(* IEC 61131-3 sources: Std_PalletMover/Class/_LMCAxisVOVMonitoring, 1 file *)

(* ---- _LMCAxisVOVMonitoring.st ---- *)
// Monitoring time (ms). If a button is not being pressed or released for a this amount of time the connection has been broken
#ifndef LMCAXIS_VOVMonitor_NoReactionTimeLimit
  #define  LMCAXIS_VOVMonitor_NoReactionTimeLimit 1000 ms
#endif

(*!
<Class
	Name               = "_LMCAxisVOVMonitoring"
	Revision           = "1.0"
	RealtimeTask       = "false"
	CyclicTask         = "false"
	BackgroundTask     = "true"
	DefBackground      = "10 ms"
	Sigmatek           = "true"
	OSInterface        = "false"
	HighPriority       = "false"
	Automatic          = "false"
	UpdateMode         = "Prescan"
	IconPath           = ".\Class\_LMCAxisVis\LMCAxis.ico"
	SharedCommandTable = "true"
	Objectsize         = "(284,120)"
	Comment            = "Class used to observe if a move hand button is still actively pressed in the VOV. If not a stop command is triggered after time LMCAXIS_VOVMonitor_NoReactionTimeLimit.">
	<Channels>
		<Server Name="ClassSvr" Visualized="false" Initialize="false" WriteProtected="true" Retentive="false"/>
		<Client Name="ToVisInt" Required="true" Internal="false"/>
	</Channels>
</Class>
*)
_LMCAxisVOVMonitoring : CLASS
  //Servers:
	ClassSvr 	: SvrChCmd_DINT;
  //Clients:
	ToVisInt 	: CltChCmd__LMCAxisVisInt;
  //Variables:
		udStartLastMove 	: UDINT;
  //Functions:
				//! <Function Comment="Background task is used to obersve if a move hand button is still pressed. If not the active move command is stopped after timeout of LMCAXIS_VOVMonitor_NoReactionTimeLimit." Name="Background"/>
	FUNCTION VIRTUAL GLOBAL Background
		VAR_INPUT
			EAX 	: UDINT;
		END_VAR
		VAR_OUTPUT
			state (EAX) 	: UDINT;
		END_VAR;
  //Tables:
	FUNCTION @STD
		VAR_OUTPUT
			ret_code	: CONFSTATES;
		END_VAR;
	FUNCTION GLOBAL TAB @CT_;
END_CLASS;

#pragma usingLtd _LMCAxisVisInt

FUNCTION VIRTUAL GLOBAL _LMCAxisVOVMonitoring::Background
	VAR_INPUT
		EAX 	: UDINT;
	END_VAR
	VAR_OUTPUT
		state (EAX) 	: UDINT;
	END_VAR

  // A move button is pressed
  if ((ToVisInt.MovNegFast.Read() <> 0) | (ToVisInt.MovNegSlow.Read() <> 0)   |
      (ToVisInt.MovPosFast.Read() <> 0) | (ToVisInt.MovPosSlow.Read() <> 0))  then

    // Get the time stamp when the button has been pressed last time
    udStartLastMove := ToVisInt.GetLastMoveTimeStamp();

  // No move button is pressed
  else
    udStartLastMove := 0;
  end_if;

  // If a button is not being pressed or released for a specified amount of time the connection has been broken
  if ((udStartLastMove <> 0) & (ops.tAbsolute - udStartLastMove > LMCAXIS_VOVMonitor_NoReactionTimeLimit)) then
    ToVisInt.StopAxis();
  end_if;

	state := READY;

END_FUNCTION
